// TIA Portal V19 export
DATA_BLOCK "DB_PAR_ID"   // DB55
{ S7_Optimized_Access := 'FALSE' }
AUTHOR : MS
// stored: AutoNumber false
   VAR RETAIN
      Anz : Int := 0;
      Offset : Int := 50;   // * Beginn Daten
      Leng : Int := 10;   // * Länge Daten
      resd : DWord := 16#0000_0000;
      resd1 : DWord := 16#0000_0000;
      resd2 : DWord := 16#0000_0000;
      resd3 : DWord := 16#0000_0000;
      resd4 : DWord := 16#0000_0000;
      resd5 : DWord := 16#0000_0000;
      resd6 : DWord := 16#0000_0000;
      resd7 : DWord := 16#0000_0000;
      resd8 : DWord := 16#0000_0000;
      resd9 : DWord := 16#0000_0000;
      resd10 : DWord := 16#0000_0000;
      Par_Config : Array[1..30] of Struct   // * Feldlänge anpassen Anzahl Positionen
         PAR1 : Byte;   // Beginn
         PAR2 : Byte;
         PAR3 : Byte;
         PAR4 : Byte;
         PAR5 : Byte;
         PAR6 : Byte;
         PAR7 : Byte;
         PAR8 : Byte;
         PAR9 : Byte;
         PAR10 : Byte;
      END_STRUCT;
   END_VAR
BEGIN
   Par_Config[1..24].PAR1 := 16#01;
   Par_Config[25..30].PAR1 := 16#00;
   Par_Config[1..30].PAR2 := 16#00;
   Par_Config[1..30].PAR3 := 16#00;
   Par_Config[1..30].PAR4 := 16#00;
   Par_Config[1..30].PAR5 := 16#00;
   Par_Config[1..30].PAR6 := 16#00;
   Par_Config[1..30].PAR7 := 16#00;
   Par_Config[1..30].PAR8 := 16#00;
   Par_Config[1..30].PAR9 := 16#00;
   Par_Config[1..30].PAR10 := 16#00;
END_DATA_BLOCK
